TYPE ST_VisMover :
STRUCT
	fPosition_X	: LREAL;
	fPosition_Y 	: LREAL;
	fPosition_Z	: LREAL;
	fPosition_A 	: LREAL;
	fPosition_B	: LREAL;
	fPosition_C	: LREAL;
	
END_STRUCT
END_TYPE

(* stored: Version 1.1.0.1, ProductVersion 3.1.4024.12
   DUT ST_VisMover: Id {25f9f235-fc97-4e1a-a85a-35ac1b912015} *)
